FUNCTION Convert_LINT_TO_ULINT : BOOL
VAR_INPUT
	in : LINT;
	out : REFERENCE TO ULINT;
END_VAR
VAR
	converted : ULINT;
END_VAR

converted := LINT_TO_ULINT(in);

IF (ULINT_TO_LINT(converted) <> in) THEN
	RETURN;
END_IF

out := converted;
Convert_LINT_TO_ULINT := TRUE;

END_FUNCTION

(* stored: Version 1.1.0.1, ProductVersion 3.1.4024.12
   POU Convert_LINT_TO_ULINT: Id {b79e1376-b346-415f-90ad-4aad0eafcec9}, SpecialFunc None *)
